FUNCTION_BLOCK FB_MQTTLog
VAR_INPUT
	Trigger:		BOOL;
	// ADSLOG_MSGTYPE_HINT or ADSLOG_MSGTYPE_WARN or ADSLOG_MSGTYPE_ERROR
	Level:			UDINT := ADSLOG_MSGTYPE_HINT;
	OnMessage: 		STRING(255) := '';
	OffMessage:		STRING(255) := '';
	OffLevel:		UDINT := 0;
END_VAR
VAR_OUTPUT
END_VAR
VAR
	LogonTrigger:	R_TRIG;
	LogoffTrigger:	F_TRIG;
	sPayloadPub:	STRING(255) := '';
END_VAR

sPayloadPub := 'log,host=CX-4E6032';
LogonTrigger(CLK := Trigger);
LogoffTrigger(CLK := Trigger);

// in case the OffLevel is not set use the default Level Value
IF OffLevel = 0 THEN
	OffLevel := Level;
END_IF
IF LogonTrigger.Q AND LEN(OnMessage)>1 THEN
	IF Level=ADSLOG_MSGTYPE_HINT THEN
		sPayloadPub := CONCAT(sPayloadPub, ',level=INFO');
	ELSIF Level=ADSLOG_MSGTYPE_WARN THEN
		sPayloadPub := CONCAT(sPayloadPub, ',level=WARNING');
	ELSE
	    sPayloadPub := CONCAT(sPayloadPub, ',level=ERROR');
	END_IF
	sPayloadPub := APPEND(sPayloadPub, ' message="', OnMessage);
	sPayloadPub := CONCAT(sPayloadPub, '"');
	MQTTCommunication.fbMqttClient.Publish(	
					sTopic:= 'RoboTel/Log', 
					pPayload:= ADR(sPayloadPub), 
					nPayloadSize:= LEN2(ADR(sPayloadPub)),
					eQoS:= TcIotMqttQos.AtMostOnceDelivery,
					bRetain:= FALSE, 
					bQueue:= FALSE );
END_IF

IF LogoffTrigger.Q AND LEN(OffMessage)>1 THEN
	IF OffLevel=ADSLOG_MSGTYPE_HINT THEN
		sPayloadPub := CONCAT(sPayloadPub, ',level=INFO');
	ELSIF OffLevel=ADSLOG_MSGTYPE_WARN THEN
		sPayloadPub := CONCAT(sPayloadPub, ',level=WARNING');
	ELSE
	    sPayloadPub := CONCAT(sPayloadPub, ',level=ERROR');
	END_IF
	
	sPayloadPub := APPEND(sPayloadPub, ' message="', OffMessage);
	sPayloadPub := CONCAT(sPayloadPub, '"');
	MQTTCommunication.fbMqttClient.Publish(	
					sTopic:= 'RoboTel/Log', 
					pPayload:= ADR(sPayloadPub), 
					nPayloadSize:= LEN2(ADR(sPayloadPub)),
					eQoS:= TcIotMqttQos.AtMostOnceDelivery,
					bRetain:= FALSE, 
					bQueue:= FALSE );
END_IF

END_FUNCTION_BLOCK

(* stored: Version 1.1.0.1, ProductVersion 3.1.4024.9
   POU FB_MQTTLog: Id {9b4576f2-4101-4b44-8d3e-ce9bf7223fb1}, SpecialFunc None *)
